(* Schneider Machine Expert - Basic project Lift, file version 2.7.0.0 *)
(* ProjectInformations: Name=New project *)

HARDWARE
  Cpu 0: TM221CE16R
  EthernetConfiguration: NetworkName=M221, IpAllocationMode=FixedAddress, IpAddress=0.0.0.0, SubnetMask=0.0.0.0
  SerialLineConfiguration: Baud=Baud19200, Parity=ParityEven, DataBits=DataBits8, StopBits=StopBits1, PhysicalMedium=PhysicalMediumRs485, TransmissionMode=TransmissionModeModbusRtu, SlaveId=1, Addressing=SlaveAddressing
  MastTask: UsePeriodScanMode=false, PeriodScan=100
  FastTask: Period=255
  CpuBehavior: StartingMode=StartAsPreviousState, AutoSaveRamOnEeprom=true, WatchdogPeriod=250

SYMBOLS  (address, symbol, comment, settings)
  %M0       OFF_ON  "Lift aan/uit"
  %M1       VERDIEPING_1  "De lift is op verdieping 1"
  %M2       VERDIEPING_2  "De lift is op verdieping 2"
  %M3       VER_1_PRESS  "Knop 1"
  %M4       OPEN_DOOR  "Deuren moeten open"
  %M5       MOTOR_OMHOOG  "Lift moet naar verdieping 2"
  %M6       VER_2_PRESS  "Knop 2"
  %M7       MOTOR_OMLAAG  "Lift moet naar beneden"
  %M8       OMHOOG
  %M9       OMLAAG
  %M10      KNIPPEREN
  %TM0      DEUR_SLUITEN  "Deur gaat dicht na 5 seconden"  [Preset=5, Base=OneSecond]
  %TM1      MOTOR_MOVING  [Preset=5, Base=OneSecond]
  %TM2        [Preset=2, Base=OneSecond]
  %TM3        [Preset=2, Base=OneSecond]
  %I0.0     ON_OFF  "Stop knop"
  %I0.2     KNIPPER  "Knipper licht"
  %I0.3     KNOP_VER_1  "Knop lift naar 1"
  %I0.4     KNOP_VER_2  "Lift naar verdieping 2"
  %Q0.0     KNIPPER_LET  "Knipper let"
  %Q0.1     MOTOR_LET  "Motor aan"
  %Q0.2     LET_1  "Lift is op verdieping 1"
  %Q0.3     LET_2  "De lift is op verdieping 2"
  %Q0.4     DOOR_OPEN  "De deuren zijn open"

POU Start lift
  (* SectionNumber=1 *)

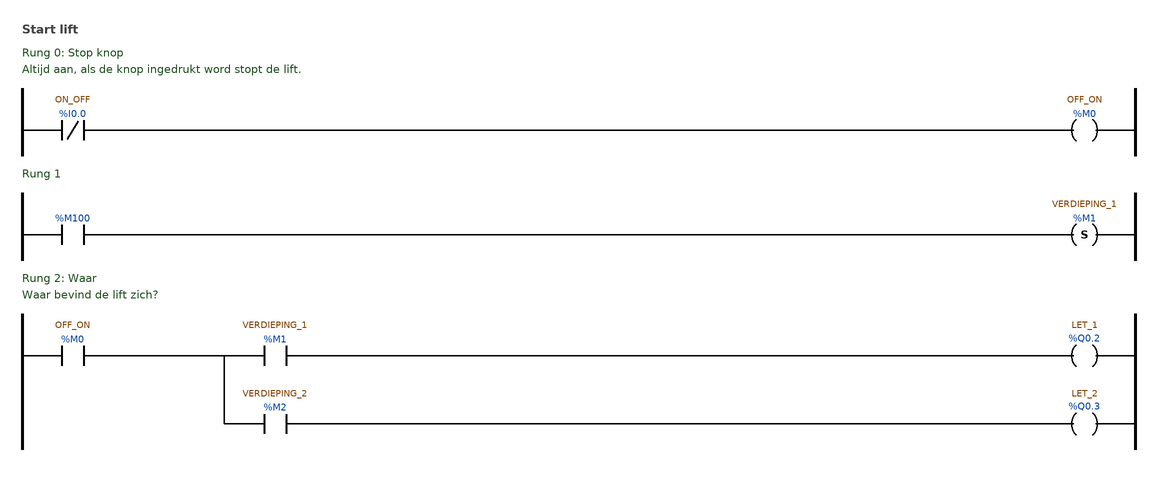

// Rung 0: Stop knop
// Altijd aan, als de knop ingedrukt word stopt de lift.
  LDN %I0.0               (* ON_OFF *)
  ST %M0                  (* OFF_ON *)
  // as ST:
  //   OFF_ON := NOT ON_OFF;

// Rung 1
  LD %M100
  S %M1                   (* VERDIEPING_1 *)
  // as ST:
  //   IF %M100 THEN VERDIEPING_1 := TRUE; END_IF;

// Rung 2: Waar
// Waar bevind de lift zich?
  LD %M0                  (* OFF_ON *)
  MPS
  AND %M1                 (* VERDIEPING_1 *)
  ST %Q0.2                (* LET_1 *)
  MPP
  AND %M2                 (* VERDIEPING_2 *)
  ST %Q0.3                (* LET_2 *)
  // as ST:
  //   LET_1 := OFF_ON AND VERDIEPING_1;
  //   LET_2 := OFF_ON AND VERDIEPING_2;

POU Deuren
  (* SectionNumber=2 *)

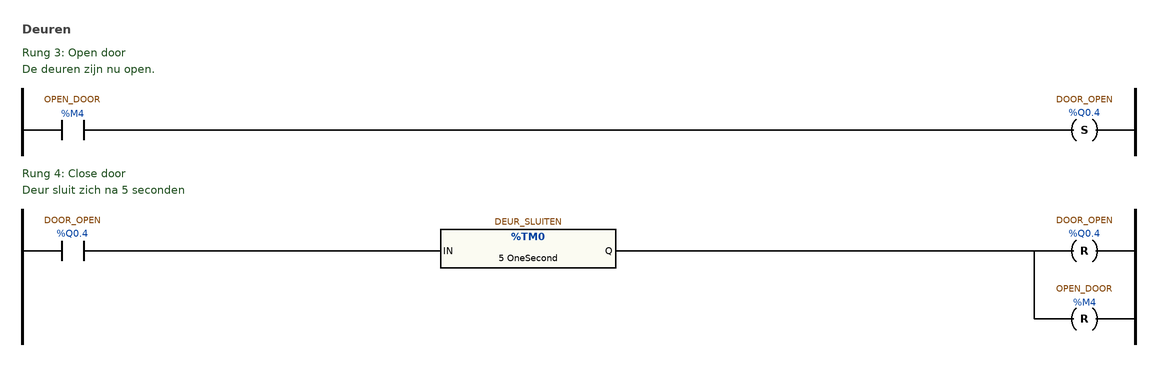

// Rung 3: Open door
// De deuren zijn nu open.
  LD %M4                  (* OPEN_DOOR *)
  S %Q0.4                 (* DOOR_OPEN *)
  // as ST:
  //   IF OPEN_DOOR THEN DOOR_OPEN := TRUE; END_IF;

// Rung 4: Close door
// Deur sluit zich na 5 seconden
  BLK %TM0                (* DEUR_SLUITEN *)
  LD %Q0.4                (* DOOR_OPEN *)
  IN
  OUT_BLK
  LD Q
  R %Q0.4                 (* DOOR_OPEN *)
  R %M4                   (* OPEN_DOOR *)
  END_BLK
  // as ST:
  //   DEUR_SLUITEN(IN := DOOR_OPEN);
  //   IF DEUR_SLUITEN.Q THEN DOOR_OPEN := FALSE; END_IF;
  //   IF DEUR_SLUITEN.Q THEN OPEN_DOOR := FALSE; END_IF;

POU Motor
  (* SectionNumber=3 *)

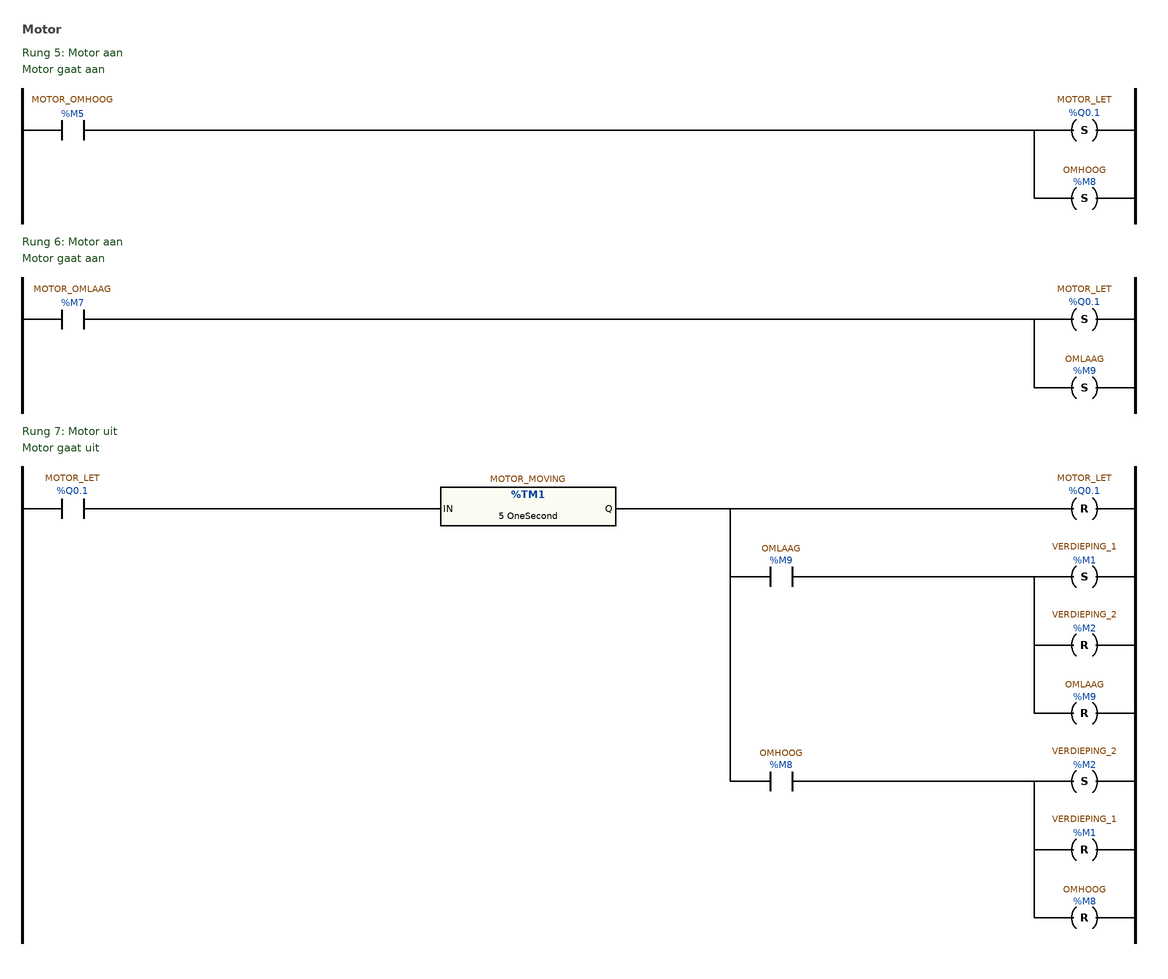

// Rung 5: Motor aan
// Motor gaat aan
  LD %M5                  (* MOTOR_OMHOOG *)
  S %Q0.1                 (* MOTOR_LET *)
  S %M8                   (* OMHOOG *)
  // as ST:
  //   IF MOTOR_OMHOOG THEN MOTOR_LET := TRUE; END_IF;
  //   IF MOTOR_OMHOOG THEN OMHOOG := TRUE; END_IF;

// Rung 6: Motor aan
// Motor gaat aan
  LD %M7                  (* MOTOR_OMLAAG *)
  S %Q0.1                 (* MOTOR_LET *)
  S %M9                   (* OMLAAG *)
  // as ST:
  //   IF MOTOR_OMLAAG THEN MOTOR_LET := TRUE; END_IF;
  //   IF MOTOR_OMLAAG THEN OMLAAG := TRUE; END_IF;

// Rung 7: Motor uit
// Motor gaat uit
  BLK %TM1                (* MOTOR_MOVING *)
  LD %Q0.1                (* MOTOR_LET *)
  IN
  OUT_BLK
  LD Q
  MPS
  R %Q0.1                 (* MOTOR_LET *)
  MRD
  AND %M9                 (* OMLAAG *)
  S %M1                   (* VERDIEPING_1 *)
  R %M2                   (* VERDIEPING_2 *)
  R %M9                   (* OMLAAG *)
  MPP
  AND %M8                 (* OMHOOG *)
  S %M2                   (* VERDIEPING_2 *)
  R %M1                   (* VERDIEPING_1 *)
  R %M8                   (* OMHOOG *)
  END_BLK
  // as ST:
  //   MOTOR_MOVING(IN := MOTOR_LET);
  //   IF MOTOR_MOVING.Q THEN MOTOR_LET := FALSE; END_IF;
  //   IF MOTOR_MOVING.Q AND OMLAAG THEN VERDIEPING_1 := TRUE; END_IF;
  //   IF MOTOR_MOVING.Q AND OMLAAG THEN VERDIEPING_2 := FALSE; END_IF;
  //   IF MOTOR_MOVING.Q AND OMLAAG THEN OMLAAG := FALSE; END_IF;
  //   IF MOTOR_MOVING.Q AND OMHOOG THEN VERDIEPING_2 := TRUE; END_IF;
  //   IF MOTOR_MOVING.Q AND OMHOOG THEN VERDIEPING_1 := FALSE; END_IF;
  //   IF MOTOR_MOVING.Q AND OMHOOG THEN OMHOOG := FALSE; END_IF;

POU Verdieping 1
  (* SectionNumber=4 *)

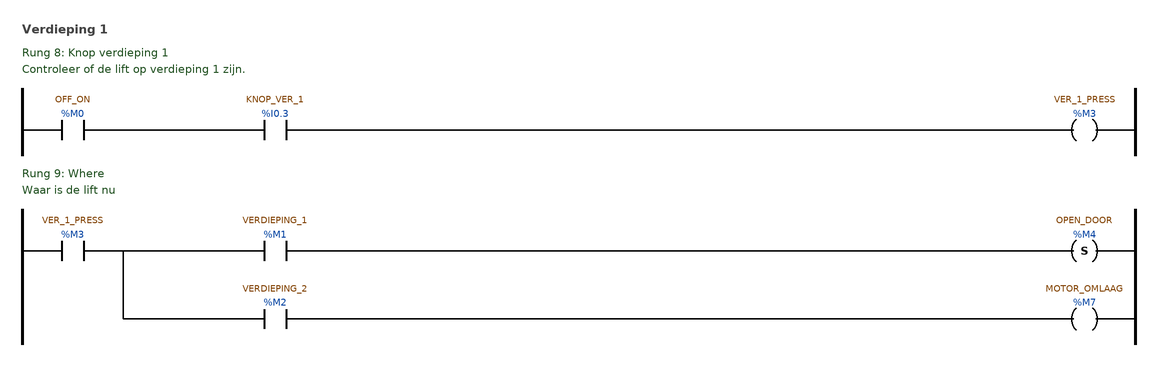

// Rung 8: Knop verdieping 1
// Controleer of de lift op verdieping 1 zijn.
  LD %M0                  (* OFF_ON *)
  AND %I0.3               (* KNOP_VER_1 *)
  ST %M3                  (* VER_1_PRESS *)
  // as ST:
  //   VER_1_PRESS := OFF_ON AND KNOP_VER_1;

// Rung 9: Where
// Waar is de lift nu
  LD %M3                  (* VER_1_PRESS *)
  MPS
  AND %M1                 (* VERDIEPING_1 *)
  S %M4                   (* OPEN_DOOR *)
  MPP
  AND %M2                 (* VERDIEPING_2 *)
  ST %M7                  (* MOTOR_OMLAAG *)
  // as ST:
  //   IF VER_1_PRESS AND VERDIEPING_1 THEN OPEN_DOOR := TRUE; END_IF;
  //   MOTOR_OMLAAG := VER_1_PRESS AND VERDIEPING_2;

POU Verdieping 2
  (* SectionNumber=5 *)

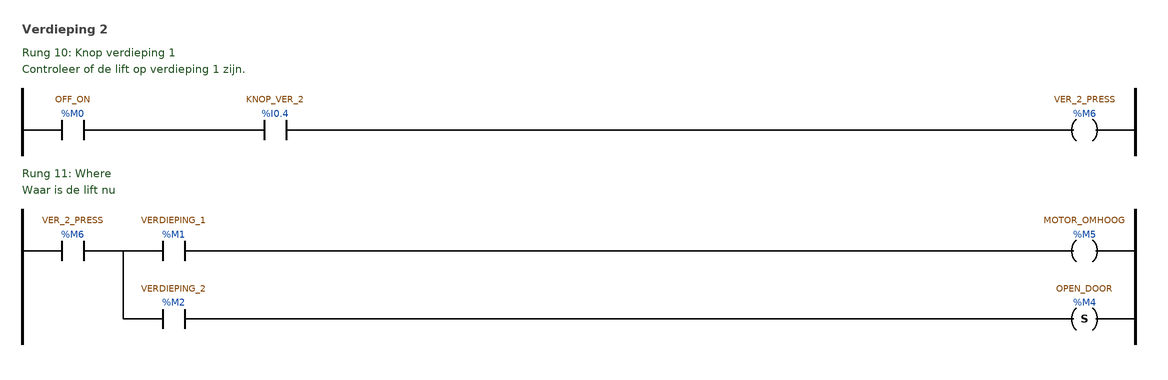

// Rung 10: Knop verdieping 1
// Controleer of de lift op verdieping 1 zijn.
  LD %M0                  (* OFF_ON *)
  AND %I0.4               (* KNOP_VER_2 *)
  ST %M6                  (* VER_2_PRESS *)
  // as ST:
  //   VER_2_PRESS := OFF_ON AND KNOP_VER_2;

// Rung 11: Where
// Waar is de lift nu
  LD %M6                  (* VER_2_PRESS *)
  MPS
  AND %M1                 (* VERDIEPING_1 *)
  ST %M5                  (* MOTOR_OMHOOG *)
  MPP
  AND %M2                 (* VERDIEPING_2 *)
  S %M4                   (* OPEN_DOOR *)
  // as ST:
  //   MOTOR_OMHOOG := VER_2_PRESS AND VERDIEPING_1;
  //   IF VER_2_PRESS AND VERDIEPING_2 THEN OPEN_DOOR := TRUE; END_IF;

POU Licht aan/uit
  (* SectionNumber=6 *)

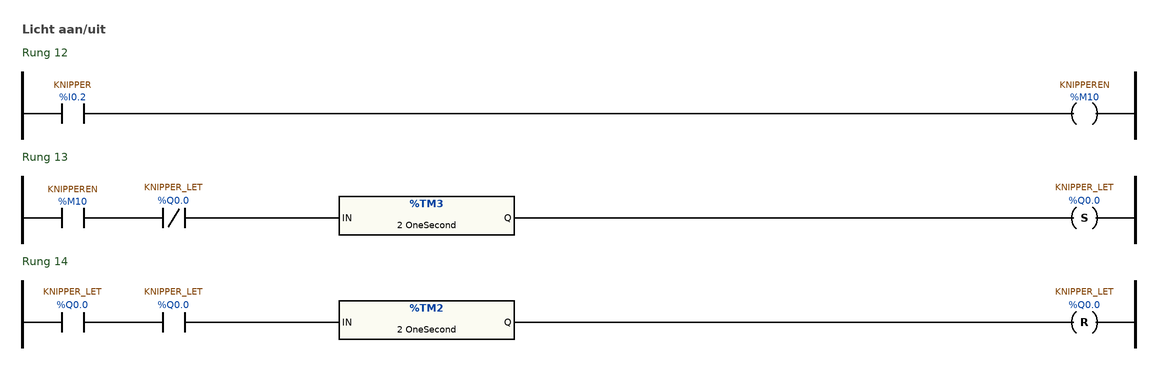

// Rung 12
  LD %I0.2                (* KNIPPER *)
  ST %M10                 (* KNIPPEREN *)
  // as ST:
  //   KNIPPEREN := KNIPPER;

// Rung 13
  BLK %TM3
  LD %M10                 (* KNIPPEREN *)
  ANDN %Q0.0              (* KNIPPER_LET *)
  IN
  OUT_BLK
  LD Q
  S %Q0.0                 (* KNIPPER_LET *)
  END_BLK
  // as ST:
  //   %TM3(IN := KNIPPEREN AND NOT KNIPPER_LET);
  //   IF %TM3.Q THEN KNIPPER_LET := TRUE; END_IF;

// Rung 14
  BLK %TM2
  LD %Q0.0                (* KNIPPER_LET *)
  AND %Q0.0               (* KNIPPER_LET *)
  IN
  OUT_BLK
  LD Q
  R %Q0.0                 (* KNIPPER_LET *)
  END_BLK
  // as ST:
  //   %TM2(IN := KNIPPER_LET AND KNIPPER_LET);
  //   IF %TM2.Q THEN KNIPPER_LET := FALSE; END_IF;
